TYPE ST_STATION_LIST_RESULT :
STRUCT
  wState    : WORD;   // wState == 0 --> all ok
  nIndex    : ULINT;
  stData    : ST_STATION_MOVER_DATA;  // copy of list entry
END_STRUCT
END_TYPE

(* stored: Version 1.1.0.1
   DUT ST_STATION_LIST_RESULT: Id {9a9316bc-78c6-4dcd-9ffd-7b75b80979b1} *)
